{attribute 'qualified_only'}
{attribute 'strict'}
{attribute 'to_string'}
TYPE E_TestEquipmentAlarmList :
(
	VerboseAlarm,
	InfoAlarm,
	WarningAlarm,
	ErrorAlarm,
	CriticalAlarm
);
END_TYPE

(* stored: Version 1.1.0.1
   DUT E_TestEquipmentAlarmList: Id {67ddde9f-8772-4ce7-884a-41098a166ea9} *)
